// TIA Portal project "washingmachine" (V12)

(* hardware
DEVICE "S7-1200 station_1"  SIMATIC 1200-Station
   slot 0: "S7-1200 rack"  Rack  V1.0
   slot 1: "PLC_1"  Unspecific CPU 1200  6ES7 2XX-XXXX-XXXX  V2.1
*)

// ===== PLC "PLC_1"  Unspecific CPU 1200 =====

VAR_GLOBAL   // PLC tag table "Washing_machine_sorting_station"
   "E-stop" AT %I0.0 : Bool;   // Emergency stop button to cut powerr from supply and circuit
   "Start PB" AT %I0.1 : Bool;   // To switch on the machine
   "Stop PB" AT %I0.2 : Bool;   // To stop the executiion if something goes wrong
   "Door Locked" AT %I0.3 : Bool;   // If the door is closed then it means that its locked
   "Inlet Valve" AT %Q0.0 : Bool;   // To let water flow into the drum
   "Cold PB" AT %I0.4 : Bool;   // Select temperature for cold wash
   "Warm PB" AT %I0.5 : Bool;   // Select temperature for warm wash
   "Cold Wash" AT %Q0.1 : Bool;
   "Warm Wash" AT %Q0.2 : Bool;
   "Drum" AT %Q0.3 : Bool;
   "Sensor S1" AT %I1.0 : Bool;   // To detect the water level in the drum
   "Sensor S2" AT %I1.1 : Bool;   // To detect if the water level in the drum
   "Red Led" AT %Q0.4 : Bool;
   "Internal Relay" AT %M100.1 : Bool;
   "Green Led" AT %Q0.5 : Bool;
   "Motor" AT %Q0.6 : Bool;   // To rotate the drum
   "Pump" AT %Q0.7 : Bool;   // To release water in the drum
   "Rinse Valve" AT %Q1.0 : Bool;
   "Door Close" AT %Q1.1 : Bool;
   "Door Open" AT %Q1.2 : Bool;
   "Level >  90" AT %I1.3 : Bool;   // To determine which sensor goes off
   "Level < 90" AT %I1.4 : Bool;   // To determine to trigger the sensor if below
   "Reset PB" AT %I0.6 : Bool;   // To reset the process and bring it to its original state
   "StartWashCycle" AT %I100.2 : Bool;
END_VAR

// folder: System blocks/Program resources

DATA_BLOCK "Motor On"   // DB1
{ S7_Optimized_Access := 'FALSE' }
AUTHOR : Simatic
FAMILY : IEC
NAME : IEC_TMR
VERSION : 1.0
// stored: InstanceOfName ?
"?"
BEGIN
END_DATA_BLOCK

DATA_BLOCK "Spin cyle"   // DB2
{ S7_Optimized_Access := 'FALSE' }
AUTHOR : Simatic
FAMILY : IEC
NAME : IEC_TMR
VERSION : 1.0
// stored: InstanceOfName ?
"?"
BEGIN
END_DATA_BLOCK

DATA_BLOCK "Motor on for spin cycle"   // DB3
{ S7_Optimized_Access := 'FALSE' }
AUTHOR : Simatic
FAMILY : IEC
NAME : IEC_TMR
VERSION : 1.0
// stored: InstanceOfName ?
"?"
BEGIN
END_DATA_BLOCK

DATA_BLOCK "drum sequnce"   // DB4
{ S7_Optimized_Access := 'FALSE' }
AUTHOR : Simatic
FAMILY : IEC
NAME : IEC_TMR
VERSION : 1.0
// stored: InstanceOfName ?
"?"
BEGIN
END_DATA_BLOCK

DATA_BLOCK "Motor Off"   // DB5
{ S7_Optimized_Access := 'FALSE' }
AUTHOR : Simatic
FAMILY : IEC
NAME : IEC_TMR
VERSION : 1.0
// stored: InstanceOfName ?
"?"
BEGIN
END_DATA_BLOCK

DATA_BLOCK "Door open sequence"   // DB6
{ S7_Optimized_Access := 'FALSE' }
AUTHOR : Simatic
FAMILY : IEC
NAME : IEC_TMR
VERSION : 1.0
// stored: InstanceOfName ?
"?"
BEGIN
END_DATA_BLOCK

// folder: (top level)

FUNCTION "Waching_machine" : Void   // FC1, LAD
{ S7_Optimized_Access := 'FALSE' }
VERSION : 0.1
// Network used to accomplish the wshing machine sequnce
BEGIN
END_FUNCTION

ORGANIZATION_BLOCK "Waching_machine_project"   // OB1, LAD, ProgramCycle
TITLE = "Main Program Sweep (Cycle)"
{ S7_Optimized_Access := 'FALSE' }
VERSION : 0.1
BEGIN

REGION Network 1
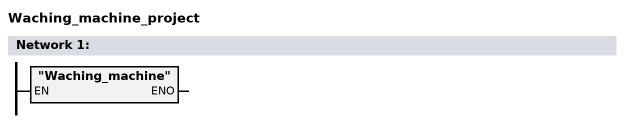
   RUNG wire#powerrail
      "Waching_machine"()
   END_RUNG
   // the same network as SCL:
   "Waching_machine"();
END_REGION
END_ORGANIZATION_BLOCK